// TIA Portal V18 export
VAR_GLOBAL   // PLC tag table "Default tag table"
   "AI8.01.01" AT %IW64 : Int;
   "AI8.01.02" AT %IW66 : Int;
   "DI8.01.01" AT %I0.0 : Bool;
   "DI8.01.02" AT %I0.1 : Bool;
   "DI8.01.03" AT %I0.2 : Bool;
   "DI8.01.04" AT %I0.3 : Bool;
   "DI8.01.05" AT %I0.4 : Bool;
   "DI8.01.06" AT %I0.5 : Bool;
   "DI8.01.07" AT %I0.6 : Bool;
   "DI8.01.08" AT %I0.7 : Bool;
   "DI8.01.09" AT %I1.0 : Bool;
   "DI8.01.10" AT %I1.1 : Bool;
   "DI8.01.11" AT %I1.2 : Bool;
   "DI8.01.12" AT %I1.3 : Bool;
   "DI8.01.13" AT %I1.4 : Bool;
   "DI8.01.14" AT %I1.5 : Bool;
   "DO8.01.01" AT %Q0.0 : Bool;
   "DO8.01.02" AT %Q0.1 : Bool;
   "DO8.01.03" AT %Q0.2 : Bool;
   "DO8.01.04" AT %Q0.3 : Bool;
   "DO8.01.05" AT %Q0.4 : Bool;
   "DO8.01.06" AT %Q0.5 : Bool;
   "DO8.01.07" AT %Q0.6 : Bool;
   "DO8.01.08" AT %Q0.7 : Bool;
   "DO8.01.09" AT %Q1.0 : Bool;
   "DO8.01.10" AT %Q1.1 : Bool;
   "AI8.02.01" AT %IW96 : Int;
   "AI8.02.02" AT %IW98 : Int;
   "AI8.02.03" AT %IW100 : Int;
   "AI8.02.04" AT %IW102 : Int;
   "AO8.03.01" AT %QW112 : Int;
   "AO8.03.02" AT %QW114 : Int;
   "AO8.03.03" AT %QW116 : Int;
   "AO8.03.04" AT %QW118 : Int;
   "DI8.04.01" AT %I16.0 : Bool;
   "DI8.04.02" AT %I16.1 : Bool;
   "DI8.04.03" AT %I16.2 : Bool;
   "DI8.04.04" AT %I16.3 : Bool;
   "DI8.04.05" AT %I16.4 : Bool;
   "DI8.04.06" AT %I16.5 : Bool;
   "DI8.04.07" AT %I16.6 : Bool;
   "DI8.04.08" AT %I16.7 : Bool;
   "DO8.04.01" AT %Q16.0 : Bool;
   "DO8.04.02" AT %Q16.1 : Bool;
   "DO8.04.03" AT %Q16.2 : Bool;
   "DO8.04.04" AT %Q16.3 : Bool;
   "DO8.04.05" AT %Q16.4 : Bool;
   "DO8.04.06" AT %Q16.5 : Bool;
   "DO8.04.07" AT %Q16.6 : Bool;
   "DO8.04.08" AT %Q16.7 : Bool;
END_VAR
